TYPE ST_ShiftRowV2 :
STRUCT
    StartMin : DINT := -1;
    DurationMin : DINT := 1440;
    ActiveDays : DINT;
END_STRUCT
END_TYPE

(* stored: Version 1.1.0.1, ProductVersion 3.1.4024.12
   DUT ST_ShiftRowV2: Id {3e46a1ef-0199-4f2b-b50b-2e4ccc014065} *)
